// TIA Portal V16 export
// export: Created 2024-09-05T17:39:24.966963Z, ExportSetting WithDefaults, DisplayName Totally Integrated Automation Portal, DisplayVersion V16 Update 6, DisplayName TIA Portal Version Control Interface, DisplayVersion V16 Update 2, DisplayName TIA Portal Openness, DisplayVersion V16 Update 6, DisplayName STEP 7 Professional, DisplayVersion V16 Update 6, DisplayName STEP 7 Safety, DisplayVersion V16, DisplayName WinCC Advanced, DisplayVersion V16 Update 6
DATA_BLOCK "6. Call_M004_NTRS_DB"   // DB2006
AUTHOR : bartz
VERSION : 0.1
// stored: AutoNumber false, DBAccessibleFromOPCUA true, InstanceOfName 6. Call_M004_NTRS, InstanceOfType FB
"6. Call_M004_NTRS"
   // VAR_INPUT
   //    nTRSTag : Bool;
   //    TIMESTAMP_IN { ExternalAccessible := 'False'; ExternalVisible := 'False'; ExternalWritable := 'False'} : WString;
   // END_VAR
   // VAR
   //    nTRSTagTemp : Bool;
   // END_VAR
BEGIN
END_DATA_BLOCK
